// TIA Portal V18 export
DATA_BLOCK "FTON_FirstTurnON"   // DB46
{ S7_Optimized_Access := 'TRUE' }
VERSION : 0.1
// stored: AutoNumber true, DBAccessibleFromOPCUA true, IsOnlyStoredInLoadMemory false, IsRetainMemResEnabled false, IsWriteProtectedInAS false, MemoryReserve 100
   VAR
      FTON_Enabled_Devices : Bool;
      FTON_Ready_Devices : Bool;
      FTON_IR_Heater_Test : Bool;
      FTON_Door_Sensor_Global : Bool := false;   // Disable Global Sensors
      FTON_Door_Sensor_FS : Bool := false;   // Disable Fluid Supply Sensor
      FTON_Data_Logging_CreateFile : Bool := false;
      FTON_Data_Logging_StartLogging : Bool;
      FTON_Turn_On_Test_Blocks : Bool;
      FTON_Run_Test_01 : Bool;
      FTON_UV_Status_Fake : Bool;
      FTON_ControlButtons : Bool := false;
      FTON_ZAxisDiagnostic : Bool := false;
   END_VAR
BEGIN
END_DATA_BLOCK
